VAR_GLOBAL CONSTANT
	cuinMaxConnections: UINT := 50;
END_VAR

(* stored: Version 1.1.0.1, ProductVersion 3.1.0.19
   GVL ACL_Const: Id {e1eec0f6-7a23-4e19-917a-fd2453668fdd} *)
